// TIA Portal V20 export
DATA_BLOCK "DriveDiagInterfaceHmi"   // DB46
TITLE = DriveDiagInterfaceHmi
AUTHOR : Siemens Digital Industries
FAMILY : LAF
NAME : LAF_DriveDiagInterfaceHmi
VERSION : 1.1
// HMI interface for drive diagnostic
// stored: MemoryReserve 100
   VAR
      diagStatus : "LAF_typeDriveDiagInterfaceHmi";
   END_VAR
BEGIN
   diagStatus.hmi.referenceDesignator := WSTRING#'';
   diagStatus.hmi.driveIndex := 0;
   diagStatus.hmi.axisStatusScreenActive := FALSE;
   diagStatus.hmi.sinaStatusScreenActive := FALSE;
   diagStatus.hmi.sinaAlarmScreenActive := FALSE;
   diagStatus.hmi.sinaEposScreenActive := FALSE;
   diagStatus.hmi.sinaSafetyScreenActive := FALSE;
   diagStatus.axis."type" := 0;
   diagStatus.axis.values.position := 0.0;
   diagStatus.axis.values.velocity := 0.0;
   diagStatus.axis.values.actualPosition := 0.0;
   diagStatus.axis.values.actualVelocity := 0.0;
   diagStatus.axis.values.actualSpeed := 0.0;
   diagStatus.axis.statusAxis.statusWord := 16#0000_0000;
   diagStatus.axis.statusAxis.statusWord2 := 16#0000_0000;
   diagStatus.axis.statusAxis.warningWord := 16#0000_0000;
   diagStatus.axis.statusAxis.errorWord := 16#0000_0000;
   diagStatus.axis.statusAxis.status.bit00_Enable := FALSE;
   diagStatus.axis.statusAxis.status.bit01_Error := FALSE;
   diagStatus.axis.statusAxis.status.bit02_RestartActive := FALSE;
   diagStatus.axis.statusAxis.status.bit03_OnlineStartValuesChanged := FALSE;
   diagStatus.axis.statusAxis.status.bit04_ControlPanelActive := FALSE;
   diagStatus.axis.statusAxis.status.bit05_HomingDone := FALSE;
   diagStatus.axis.statusAxis.status.bit06_Done := FALSE;
   diagStatus.axis.statusAxis.status.bit07_Standstill := FALSE;
   diagStatus.axis.statusAxis.status.bit08_PositioningCommand := FALSE;
   diagStatus.axis.statusAxis.status.bit09_JogCommand := FALSE;
   diagStatus.axis.statusAxis.status.bit10_VelocityCommand := FALSE;
   diagStatus.axis.statusAxis.status.bit11_HomingCommand := FALSE;
   diagStatus.axis.statusAxis.status.bit12_ConstantVelocity := FALSE;
   diagStatus.axis.statusAxis.status.bit13_Accelerating := FALSE;
   diagStatus.axis.statusAxis.status.bit14_Decelerating := FALSE;
   diagStatus.axis.statusAxis.status.bit15_SWLimitMinActive := FALSE;
   diagStatus.axis.statusAxis.status.bit16_SWLimitMaxActive := FALSE;
   diagStatus.axis.statusAxis.status.bit17_HWLimitMinActive := FALSE;
   diagStatus.axis.statusAxis.status.bit18_HWLimitMaxActive := FALSE;
   diagStatus.axis.statusAxis.status.bit19_Reserved := FALSE;
   diagStatus.axis.statusAxis.status.bit20_Reserved := FALSE;
   diagStatus.axis.statusAxis.status.bit21_Synchronizing := FALSE;
   diagStatus.axis.statusAxis.status.bit22_Synchronous := FALSE;
   diagStatus.axis.statusAxis.status.bit23_SuperimposedMotionCommand := FALSE;
   diagStatus.axis.statusAxis.status.bit24_PhasingCommand := FALSE;
   diagStatus.axis.statusAxis.status.bit25_AxisSimulation := FALSE;
   diagStatus.axis.statusAxis.status.bit26_TorqueLimitingCommand := FALSE;
   diagStatus.axis.statusAxis.status.bit27_InLimitation := FALSE;
   diagStatus.axis.statusAxis.status.bit28_NonPositionControlled := FALSE;
   diagStatus.axis.statusAxis.status.bit29_KinematicsMotionCommand := FALSE;
   diagStatus.axis.statusAxis.status.bit30_InClamping := FALSE;
   diagStatus.axis.statusAxis.status.bit31_MotionInCommand := FALSE;
   diagStatus.axis.statusAxis.status2.bit00_StopCommand := FALSE;
   diagStatus.axis.statusAxis.status2.bit01_DesynchronizingCommand := FALSE;
   diagStatus.axis.statusAxis.status2.bit02_PassingBacklash := FALSE;
   diagStatus.axis.statusAxis.status2.bit03_PhasingCommandWaiting := FALSE;
   diagStatus.axis.statusAxis.status2.bit04_OffsetCommand := FALSE;
   diagStatus.axis.statusAxis.status2.bit05_OffsetCommandWaiting := FALSE;
   diagStatus.axis.statusAxis.status2.bit06_MotionInSuperimposedCommand := FALSE;
   diagStatus.axis.statusAxis.status2.bit07_HaltSuperimposedCommand := FALSE;
   diagStatus.axis.statusAxis.status2.bit08_Reserved := FALSE;
   diagStatus.axis.statusAxis.status2.bit09_Reserved := FALSE;
   diagStatus.axis.statusAxis.status2.bit10_Reserved := FALSE;
   diagStatus.axis.statusAxis.status2.bit11_Reserved := FALSE;
   diagStatus.axis.statusAxis.status2.bit12_Reserved := FALSE;
   diagStatus.axis.statusAxis.status2.bit13_Reserved := FALSE;
   diagStatus.axis.statusAxis.status2.bit14_Reserved := FALSE;
   diagStatus.axis.statusAxis.status2.bit15_Reserved := FALSE;
   diagStatus.axis.statusAxis.status2.bit16_Reserved := FALSE;
   diagStatus.axis.statusAxis.status2.bit17_Reserved := FALSE;
   diagStatus.axis.statusAxis.status2.bit18_Reserved := FALSE;
   diagStatus.axis.statusAxis.status2.bit19_Reserved := FALSE;
   diagStatus.axis.statusAxis.status2.bit20_Reserved := FALSE;
   diagStatus.axis.statusAxis.status2.bit21_Reserved := FALSE;
   diagStatus.axis.statusAxis.status2.bit22_Reserved := FALSE;
   diagStatus.axis.statusAxis.status2.bit23_Reserved := FALSE;
   diagStatus.axis.statusAxis.status2.bit24_Reserved := FALSE;
   diagStatus.axis.statusAxis.status2.bit25_Reserved := FALSE;
   diagStatus.axis.statusAxis.status2.bit26_Reserved := FALSE;
   diagStatus.axis.statusAxis.status2.bit27_Reserved := FALSE;
   diagStatus.axis.statusAxis.status2.bit28_Reserved := FALSE;
   diagStatus.axis.statusAxis.status2.bit29_Reserved := FALSE;
   diagStatus.axis.statusAxis.status2.bit30_Reserved := FALSE;
   diagStatus.axis.statusAxis.status2.bit31_Reserved := FALSE;
   diagStatus.axis.statusAxis.warning.bit00_SystemWarning := FALSE;
   diagStatus.axis.statusAxis.warning.bit01_ConfigWarning := FALSE;
   diagStatus.axis.statusAxis.warning.bit02_UserWarning := FALSE;
   diagStatus.axis.statusAxis.warning.bit03_CommandNotAccepted := FALSE;
   diagStatus.axis.statusAxis.warning.bit04_DriveWarning := FALSE;
   diagStatus.axis.statusAxis.warning.bit05_SensorWarning := FALSE;
   diagStatus.axis.statusAxis.warning.bit06_DynamicWarning := FALSE;
   diagStatus.axis.statusAxis.warning.bit07_CommunicationWarning := FALSE;
   diagStatus.axis.statusAxis.warning.bit08_SWLimitMin := FALSE;
   diagStatus.axis.statusAxis.warning.bit09_SWLimitMax := FALSE;
   diagStatus.axis.statusAxis.warning.bit10_HomingWarning := FALSE;
   diagStatus.axis.statusAxis.warning.bit11_FollowingErrorWarning := FALSE;
   diagStatus.axis.statusAxis.warning.bit12_PositioningWarning := FALSE;
   diagStatus.axis.statusAxis.warning.bit13_PeripheralWarning := FALSE;
   diagStatus.axis.statusAxis.warning.bit14_SynchronousWarning := FALSE;
   diagStatus.axis.statusAxis.warning.bit15_AdaptionWarning := FALSE;
   diagStatus.axis.statusAxis.warning.bit16_Reserved := FALSE;
   diagStatus.axis.statusAxis.warning.bit17_Reserved := FALSE;
   diagStatus.axis.statusAxis.warning.bit18_Reserved := FALSE;
   diagStatus.axis.statusAxis.warning.bit19_Reserved := FALSE;
   diagStatus.axis.statusAxis.warning.bit20_Reserved := FALSE;
   diagStatus.axis.statusAxis.warning.bit21_Reserved := FALSE;
   diagStatus.axis.statusAxis.warning.bit22_Reserved := FALSE;
   diagStatus.axis.statusAxis.warning.bit23_Reserved := FALSE;
   diagStatus.axis.statusAxis.warning.bit24_Reserved := FALSE;
   diagStatus.axis.statusAxis.warning.bit25_Reserved := FALSE;
   diagStatus.axis.statusAxis.warning.bit26_Reserved := FALSE;
   diagStatus.axis.statusAxis.warning.bit27_Reserved := FALSE;
   diagStatus.axis.statusAxis.warning.bit28_Reserved := FALSE;
   diagStatus.axis.statusAxis.warning.bit29_Reserved := FALSE;
   diagStatus.axis.statusAxis.warning.bit30_Reserved := FALSE;
   diagStatus.axis.statusAxis.warning.bit31_Reserved := FALSE;
   diagStatus.axis.statusAxis.error.bit00_SystemFault := FALSE;
   diagStatus.axis.statusAxis.error.bit01_ConfigFault := FALSE;
   diagStatus.axis.statusAxis.error.bit02_UserFault := FALSE;
   diagStatus.axis.statusAxis.error.bit03_CommandNotAccepted := FALSE;
   diagStatus.axis.statusAxis.error.bit04_DriveFault := FALSE;
   diagStatus.axis.statusAxis.error.bit05_SensorFault := FALSE;
   diagStatus.axis.statusAxis.error.bit06_DynamicError := FALSE;
   diagStatus.axis.statusAxis.error.bit07_CommunicationFault := FALSE;
   diagStatus.axis.statusAxis.error.bit08_SWLimit := FALSE;
   diagStatus.axis.statusAxis.error.bit09_HWLimit := FALSE;
   diagStatus.axis.statusAxis.error.bit10_HomingError := FALSE;
   diagStatus.axis.statusAxis.error.bit11_FollowingErrorFault := FALSE;
   diagStatus.axis.statusAxis.error.bit12_PositioningFault := FALSE;
   diagStatus.axis.statusAxis.error.bit13_PeripheralError := FALSE;
   diagStatus.axis.statusAxis.error.bit14_SynchronousError := FALSE;
   diagStatus.axis.statusAxis.error.bit15_AdaptionError := FALSE;
   diagStatus.axis.statusAxis.error.bit16_Reserved := FALSE;
   diagStatus.axis.statusAxis.error.bit17_Reserved := FALSE;
   diagStatus.axis.statusAxis.error.bit18_Reserved := FALSE;
   diagStatus.axis.statusAxis.error.bit19_Reserved := FALSE;
   diagStatus.axis.statusAxis.error.bit20_Reserved := FALSE;
   diagStatus.axis.statusAxis.error.bit21_Reserved := FALSE;
   diagStatus.axis.statusAxis.error.bit22_Reserved := FALSE;
   diagStatus.axis.statusAxis.error.bit23_Reserved := FALSE;
   diagStatus.axis.statusAxis.error.bit24_Reserved := FALSE;
   diagStatus.axis.statusAxis.error.bit25_Reserved := FALSE;
   diagStatus.axis.statusAxis.error.bit26_Reserved := FALSE;
   diagStatus.axis.statusAxis.error.bit27_Reserved := FALSE;
   diagStatus.axis.statusAxis.error.bit28_Reserved := FALSE;
   diagStatus.axis.statusAxis.error.bit29_Reserved := FALSE;
   diagStatus.axis.statusAxis.error.bit30_Reserved := FALSE;
   diagStatus.axis.statusAxis.error.bit31_Reserved := FALSE;
   diagStatus.axis.statusAxis.errorDetail.number := 0;
   diagStatus.axis.statusAxis.errorDetail.reaction := 0;
   diagStatus.axis.statusSensor.operativeSensor := 1;
   diagStatus.axis.statusSensor.sensor[1..4].state := 0;
   diagStatus.axis.statusSensor.sensor[1..4].communicationOK := FALSE;
   diagStatus.axis.statusSensor.sensor[1..4].error := FALSE;
   diagStatus.axis.statusSensor.sensor[1..4].control := FALSE;
   diagStatus.axis.statusSensor.sensor[1..4].position := 0.0;
   diagStatus.axis.statusSensor.sensor[1..4].velocity := 0.0;
   diagStatus.axis.statusSensor.sensor[1..4].adaptionState := 0;
   diagStatus.axis.statusSensor.sensor[1..4].adjusted := 0;
   diagStatus.axis.statusPositioning.targetPosition := 0.0;
   diagStatus.axis.statusPositioning.followingError := 0.0;
   diagStatus.axis.units.lengthUnit := 0;
   diagStatus.axis.units.velocityUnit := 0;
   diagStatus.sina.sinaType := 0;
   diagStatus.sina.controlWord := 16#0000;
   diagStatus.sina.statusWord := 16#0000;
   diagStatus.sina.telegramNo := 0;
   diagStatus.sina.eposStatusWord1 := 16#0000;
   diagStatus.sina.eposStatusWord2 := 16#0000;
   diagStatus.sina.operatingDisplay := 0;
   diagStatus.sina.override := 0.0;
   diagStatus.sina.posSetValue := 0.0;
   diagStatus.sina.posActValue := 0.0;
   diagStatus.sina.velSetValue := 0.0;
   diagStatus.sina.velActValue := 0.0;
   diagStatus.sina.lengthUnit := 0;
   diagStatus.sina.velocityUnit := 0;
   diagStatus.sina.residualDistance := 0.0;
   diagStatus.sina.followingError := 0.0;
   diagStatus.sina.posControlWord := 16#0000;
   diagStatus.sina.posStatusWord := 16#0000;
   diagStatus.sina.blockSelected := 0;
   diagStatus.sina.blockActive := 0;
   diagStatus.sina.mdiPosSetValue := 0.0;
   diagStatus.sina.faultCode[0..7] := 16#0000;
   diagStatus.sina.alarmCode[0..3] := 16#0000;
   diagStatus.sina.speedSetValue := 0.0;
   diagStatus.sina.speedActValue := 0.0;
   diagStatus.sina.safetyStatusWord := 16#0000;
END_DATA_BLOCK
